// TIA Portal V20 export
FUNCTION_BLOCK "FB_WorkingModes"   // FB56, SCL
{ S7_Optimized_Access := 'TRUE' }
// stored: MemoryReserve 100, SetENOAutomatically false
   VAR_INPUT
      iChangeModeEnable : Bool;
   END_VAR
   VAR_IN_OUT
      ioEmptyingReq : Bool;
      ioAutoReq : Bool;
      ioSemiAutoReq : Bool;
      ioManuReq : Bool;
   END_VAR
   VAR
      sRT_Filling : R_TRIG;
      sRT_Normal { S7_SetPoint := 'True'} : R_TRIG;
      sRT_Emptying { S7_SetPoint := 'True'} : R_TRIG;
      sFT_Emptying { S7_SetPoint := 'True'} : F_TRIG;
      sRT_Auto { S7_SetPoint := 'True'} : R_TRIG;
      sRT_SemiAuto { S7_SetPoint := 'True'} : R_TRIG;
      sRT_Manu { S7_SetPoint := 'True'} : R_TRIG;
      sFilling { S7_SetPoint := 'True'} : Bool;
      sNormal : Bool;
      sEmptying : Bool;
      sAuto : Bool;
      sSemiAuto : Bool;
      sManu : Bool;
      sOnePiece : Bool;
      sDryRun : Bool;
   END_VAR
BEGIN
   REGION Description header 
       //==================================================================================
       // POSALUX Swiss SA / (C) Copyright 2025
       //----------------------------------------------------------------------------------
       // Title: FB_WorkingModes
       // Comment/Function: 
       // Author: Fabien WALDT
       // Engineering: TIA Portal v17
       //----------------------------------------------------------------------------------
       // Change log table:
       // Version  | Date     | Expert in charge | Changes applied
       // ---------|----------|------------------|-----------------------------------------
       // 00.00.01 | 20251218 | WFA              | First released version
       // =================================================================================
   END_REGION

   REGION Filling - Normal - Emptying
       #sRT_Emptying(CLK := #ioEmptyingReq);
       #sFT_Emptying(CLK := #ioEmptyingReq);

       #sRT_Filling(CLK := ("DB_LoaderShuttle1".sMain.iJobReq OR "DB_LoaderShuttle2".sMain.iJobReq)
                    AND "DB_PartManagement".sPosition.sMachineEmpty AND NOT #sEmptying);

       #sRT_Normal(CLK := (("DB_LoaderShuttle1".sMain.iJobReq OR "DB_LoaderShuttle2".sMain.iJobReq)
                   AND NOT "DB_PartManagement".sPosition.sMachineEmpty
                   AND NOT #sFilling)
                   OR ("DB_PartManagement".sPosition.sFixture.Drilled.Presence.Part AND NOT #sNormal AND NOT #sEmptying)
                   OR #sFT_Emptying.Q);

       IF #sRT_Filling.Q THEN
           #sFilling := TRUE;
           #sNormal := FALSE;
           #sEmptying := FALSE;
       END_IF;

       IF #sRT_Normal.Q THEN
           #sFilling := FALSE;
           #sNormal := TRUE;
           #sEmptying := FALSE;
       END_IF;

       IF #sRT_Emptying.Q THEN
           #sFilling := FALSE;
           #sNormal := FALSE;
           #sEmptying := TRUE;
       END_IF;
   END_REGION

   REGION Auto - Semi Auto - Manu
       #sRT_Auto(CLK := #ioAutoReq OR (NOT #sAuto AND NOT #sSemiAuto AND NOT #sManu));
       #sRT_SemiAuto(CLK := #ioSemiAutoReq);
       #sRT_Manu(CLK := #ioManuReq);

       IF #iChangeModeEnable THEN
           IF #sRT_Auto.Q THEN
               #sAuto := TRUE;
               #sSemiAuto := FALSE;
               #sManu := FALSE;
           ELSIF #sRT_SemiAuto.Q THEN
               #sAuto := FALSE;
               #sSemiAuto := TRUE;
               #sManu := FALSE;
           ELSIF #sRT_Manu.Q THEN
               #sAuto := FALSE;
               #sSemiAuto := FALSE;
               #sManu := TRUE;
           END_IF;
       END_IF;

       #ioAutoReq := FALSE;
       #ioSemiAutoReq := FALSE;
       #ioManuReq := FALSE;
   END_REGION
END_FUNCTION_BLOCK
